FUNCTION_BLOCK FB_MUX
VAR_INPUT
	in1,in2:INT;
END_VAR
VAR_OUTPUT
	out:INT;
END_VAR
VAR
END_VAR

out:=in1*in2;

END_FUNCTION_BLOCK

(* stored: Version 1.1.0.1, ProductVersion 3.1.4024.11
   POU FB_MUX: Id {a133e9c4-d39f-46fb-b382-f88dd4608554}, SpecialFunc None *)
